RoboDK station: Tarea3Definitiva2_IsabellaCeballos.rdk

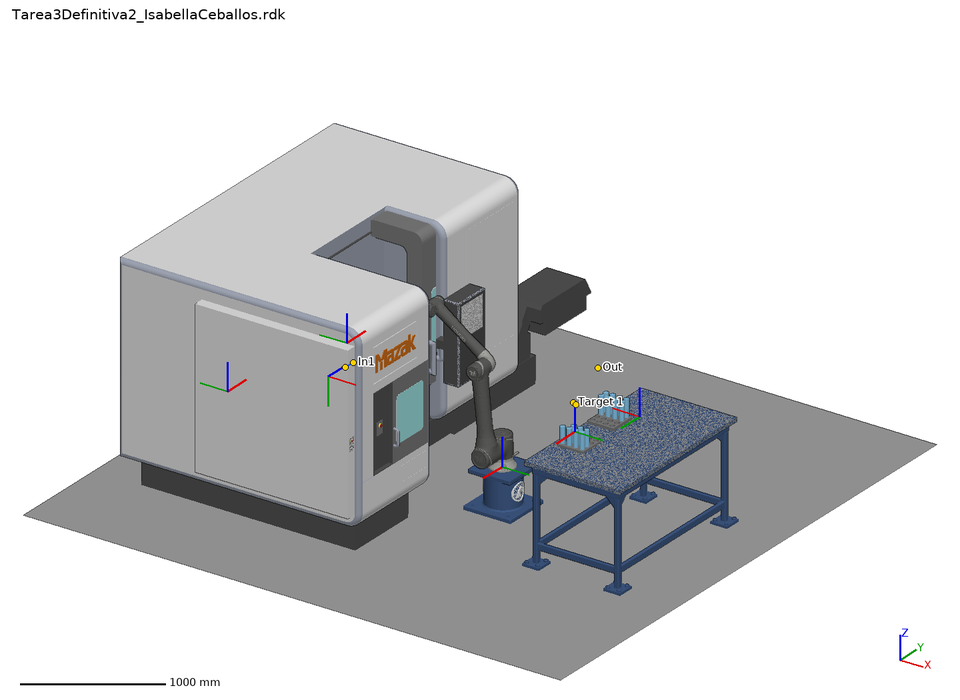
[picture v0: the station drawn from its stored meshes, robots at their saved joint values, targets as dots, program paths as lines]
Station Tarea3Definitiva2_IsabellaCeballos (saved by RoboDK 5.5.1). Poses are relative to the parent item; angles as X-Y-Z fixed-axis rotations.
Station parameters (name, value as stored): TAGS, ['Machine Tending', 'CNC']
  - frame Omron TM12X Base at (300, 0, 70) mm, rotated rx 0 ry 0 rz -90 deg
    - robot Omron TM12X: 6 axes, payload 12 kg, reach 1300 mm, repeatability 0.1 mm, weight 33.3 kg
        modified DH rows (alpha deg, a mm, theta deg, d mm): 0, 0, 0, 165.2; 90, 0, 90, 0; 0, 636.1, 0, 0; 0, 557.9, -90, 156.3; -90, 0, 0, 106; 90, 0, 180, 113.15
        joint limits [-360, -360, -163, -360, -360, -360] to [360, 360, 163, 360, 360, 360]; home [0, 0, 90, -90, 90, 0]; saved at [90.435, -6.151, -48.82, -37.474, -88.325, 69.903]
      - tool g1, TCP at (0, 0, 130) mm, size 134.4 x 157.6 x 75 mm
        - object Part 8 at (4.25, 9.04, 154.7) mm, rotated rx 177.54 ry -1.66 rz -69.47 deg, size 40 x 40 x 150 mm, geometry from Part.step
      - tool RobotiQ 2F-85 Gripper (Open), TCP at (0, 0, 130) mm, size 147.4 x 146.8 x 75 mm
    - object Pedestal H12in (Type 1) at (0, 10, -300) mm, size 400 x 400 x 304.8 mm, geometry from Pedestal-H12in-Type-1.sld
  - frame Mazak Lathe Base at (-1000, 0, 650) mm, rotated rx 0 ry 0 rz 90 deg
    - robot Mazak Lathe: 1 axes
        modified DH rows (alpha deg, a mm, theta deg, d mm): 0, 0, 0, 0 linear
        base shift (0, 0, 0) mm, rotated rx 0 ry 90 rz 0 deg
        joint limits [0] to [700]; home [0]; saved at [691]
    - frame Lathe at (-368.68, -104.77, -79.13) mm, rotated rx -90 ry 0 rz -90 deg
  - frame Input at (1010, -140, 590) mm, rotated rx 0 ry 0 rz -90 deg
    - object Part Matrix at (0, 0, 0) mm, size 220 x 220 x 25 mm, geometry from Part Matrix.step
    - target Target 1 (Cartesian target) at (-26.53, -36.52, 202.61) mm, rotated rx -177.37 ry 1.91 rz -69.45 deg; joints [247.43, -1, -72.52, -13.29, -90.61, 226.91] of Omron TM12X
    - object Part 6 at (137.5, 137.5, -20) mm, size 40 x 40 x 150 mm, geometry from Part.step
    - object Part 1 at (192.5, 192.5, -20) mm, size 40 x 40 x 150 mm, geometry from Part.step
    - object Part 5 at (137.5, 192.5, -20) mm, size 40 x 40 x 150 mm, geometry from Part.step
    - object Part 7 at (137.5, 82.5, -20) mm, size 40 x 40 x 150 mm, geometry from Part.step
    - object Part 4 at (192.5, 27.5, -20) mm, rotated rx 0 ry 0 rz -180 deg, size 40 x 40 x 150 mm, geometry from Part.step
    - object Part 3 at (192.5, 82.5, -20) mm, rotated rx 0 ry 0 rz -180 deg, size 40 x 40 x 150 mm, geometry from Part.step
    - object Part 2 at (192.5, 137.5, -20) mm, rotated rx 0 ry 0 rz -180 deg, size 40 x 40 x 150 mm, geometry from Part.step
    - target Home (Cartesian target) at (28, 28, 225) mm, rotated rx -177.37 ry 1.91 rz -69.45 deg; joints [245.421, -8.702, -61.622, -16.467, -90.498, 224.904] of Omron TM12X
    - target Out (Cartesian target) at (-404.5, -94.61, 298.15) mm, rotated rx 179.32 ry 1.81 rz -82.53 deg; joints [279.536, -58.254, 58.657, -88.574, -89.388, -87.935] of Omron TM12X
  - frame Output at (1250, 290, 600) mm, rotated rx 0 ry 0 rz -180 deg
    - object Part Matrix at (47.8, 28.1, 0) mm, size 220 x 220 x 25 mm, geometry from Part Matrix.step
    - object Part 16 at (75.39, 55.49, -8.13) mm, rotated rx 0 ry 0 rz 90 deg, size 40 x 40 x 150 mm, geometry from Part.step
    - object Part 15 at (132.39, 55.49, -8.13) mm, rotated rx 0 ry 0 rz 90 deg, size 40 x 40 x 150 mm, geometry from Part.step
    - object Part 14 at (189.39, 55.49, -8.13) mm, rotated rx 0 ry 0 rz 90 deg, size 40 x 40 x 150 mm, geometry from Part.step
    - object Part 13 at (246.39, 55.49, -8.13) mm, rotated rx 0 ry 0 rz 90 deg, size 40 x 40 x 150 mm, geometry from Part.step
    - object Part 12 at (75.39, 110.49, -8.13) mm, rotated rx 0 ry 0 rz 90 deg, size 40 x 40 x 150 mm, geometry from Part.step
    - object Part 11 at (132.39, 110.49, -8.13) mm, rotated rx 0 ry 0 rz 90 deg, size 40 x 40 x 150 mm, geometry from Part.step
    - object Part 10 at (189.39, 110.49, -8.13) mm, rotated rx 0 ry 0 rz 90 deg, size 40 x 40 x 150 mm, geometry from Part.step
    - object Part 9 at (246.39, 110.49, -8.13) mm, rotated rx 0 ry 0 rz 90 deg, size 40 x 40 x 150 mm, geometry from Part.step
  - frame World at (-2000, 0, 0) mm, rotated rx 0 ry 0 rz 90 deg
    - object Floor at (250, -1940, -230) mm, size 4500 x 4500 x 0 mm, geometry from Floor (2).sld
    - object Table 1400x800x800mm at (-340, -3360, 570) mm, size 1420 x 820 x 800 mm, geometry from Table-1400x800x800mm.sld
    - target OpenDoor (Cartesian target) at (700, -1000, 650) mm; joints [700] of Mazak Lathe
    - target CloseDoor (Cartesian target) at (0, -1000, 650) mm; joints [0] of Mazak Lathe
    - target In1 (Cartesian target) at (-137.95, -1150.25, 595.88) mm, rotated rx -86.34 ry 2.11 rz 94.34 deg; joints [77.244, -89.992, 25.646, 51.981, -342.661, 170.292] of Omron TM12X
    - target In2 (Cartesian target) at (-206.56, -1130.76, 584.67) mm, rotated rx -87.8 ry 7.87 rz 92.76 deg; joints [-84.147, 66.082, 6.025, 75.079, -175.968, 40.623] of Omron TM12X
  - program atach (1 instructions, listed below)
  - program detach (1 instructions, listed below)
  - program init (1 instructions, listed below)
  - program OpenDoor (2 instructions, listed below)
  - program CloseDoor (2 instructions, listed below)
  - program GoHome (3 instructions, listed below)
  - program Go_Out (3 instructions, listed below)
  - program Main_Program (496 instructions, listed below)
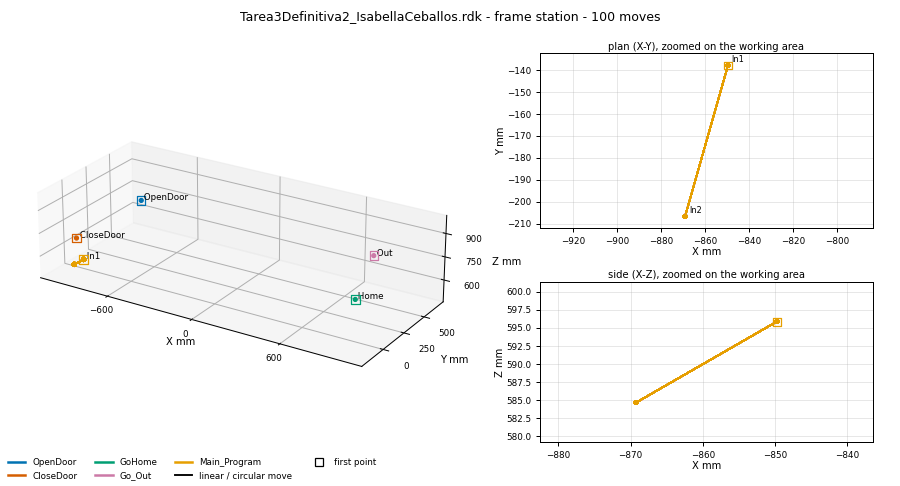
[picture p0: tool path of Tarea3Definitiva2_IsabellaCeballos.rdk in frame station, 100 of 276 moves have a stored position in this frame; points joined in program order, loops and branches not executed]

--- program atach (robot Omron TM12X) ---
  Adjuntar a g1

--- program detach (robot Omron TM12X) ---
  Separar de g1

--- program init (robot Omron TM12X) ---
  Reemplazar objetos

--- program OpenDoor (robot Mazak Lathe) ---
  Est. Ref.: World
  MoveJ (OpenDoor)

--- program CloseDoor (robot Mazak Lathe) ---
  Est. Ref.: World
  MoveJ (CloseDoor)

--- program GoHome (robot Omron TM12X) ---
  Est. Ref.: Input
  Est. herr: g1
  MoveJ (Home)

--- program Go_Out (robot Omron TM12X) ---
  Est. Ref.: Input
  Est. herr: g1
  MoveJ (Out)

--- program Main_Program (robot Omron TM12X) ---
  Est. Ref.: Input
  MoveJ (Auto Up_Pick 1) [its target is no longer in the station]
  MoveL (Auto Pick 1) [its target is no longer in the station]
  Llamar atach
  MoveL (Auto Up_Pick 1) [its target is no longer in the station]
  MoveL (Auto Transition 1) [its target is no longer in the station]
  MoveJ (Auto Transition 2) [its target is no longer in the station]
  Llamar OpenDoor
  Est. Ref.: World
  MoveJ (In1)
  MoveL (In2)
  Llamar detach
  MoveL (In1)
  Est. Ref.: Input
  MoveJ (Auto Transition 2) [its target is no longer in the station]
  Llamar CloseDoor
  Llamar OpenDoor
  Est. Ref.: World
  MoveJ (In1)
  MoveL (In2)
  Llamar atach
  MoveL (In1)
  Est. Ref.: Input
  MoveJ (Auto Transition 2) [its target is no longer in the station]
  Llamar CloseDoor
  MoveL (Auto Transition 1) [its target is no longer in the station]
  Llamar Go_Out
  MoveJ (Auto Drop_Up 1) [its target is no longer in the station]
  MoveL (Auto Drop 1) [its target is no longer in the station]
  Llamar detach
  MoveL (Auto Drop_Up 1) [its target is no longer in the station]
  Est. Ref.: Input
  MoveJ (Auto Up_Pick 2) [its target is no longer in the station]
  MoveL (Auto Pick 2) [its target is no longer in the station]
  Llamar atach
  MoveL (Auto Up_Pick 2) [its target is no longer in the station]
  MoveL (Auto Transition 1) [its target is no longer in the station]
  MoveJ (Auto Transition 2) [its target is no longer in the station]
  Llamar OpenDoor
  Est. Ref.: World
  MoveJ (In1)
  MoveL (In2)
  Llamar detach
  MoveL (In1)
  Est. Ref.: Input
  MoveJ (Auto Transition 2) [its target is no longer in the station]
  Llamar CloseDoor
  Llamar OpenDoor
  Est. Ref.: World
  MoveJ (In1)
  MoveL (In2)
  Llamar atach
  MoveL (In1)
  Est. Ref.: Input
  MoveJ (Auto Transition 2) [its target is no longer in the station]
  Llamar CloseDoor
  MoveL (Auto Transition 1) [its target is no longer in the station]
  Llamar Go_Out
  MoveJ (Auto Drop_Up 2) [its target is no longer in the station]
  MoveL (Auto Drop 2) [its target is no longer in the station]
  Llamar detach
  MoveL (Auto Drop_Up 2) [its target is no longer in the station]
  Est. Ref.: Input
  MoveJ (Auto Up_Pick 3) [its target is no longer in the station]
  MoveL (Auto Pick 3) [its target is no longer in the station]
  Llamar atach
  MoveL (Auto Up_Pick 3) [its target is no longer in the station]
  MoveL (Auto Transition 1) [its target is no longer in the station]
  MoveJ (Auto Transition 2) [its target is no longer in the station]
  Llamar OpenDoor
  Est. Ref.: World
  MoveJ (In1)
  MoveL (In2)
  Llamar detach
  MoveL (In1)
  Est. Ref.: Input
  MoveJ (Auto Transition 2) [its target is no longer in the station]
  Llamar CloseDoor
  Llamar OpenDoor
  Est. Ref.: World
  MoveJ (In1)
  MoveL (In2)
  Llamar atach
  MoveL (In1)
  Est. Ref.: Input
  MoveJ (Auto Transition 2) [its target is no longer in the station]
  Llamar CloseDoor
  MoveL (Auto Transition 1) [its target is no longer in the station]
  Llamar Go_Out
  MoveJ (Auto Drop_Up 3) [its target is no longer in the station]
  MoveL (Auto Drop 3) [its target is no longer in the station]
  Llamar detach
  MoveL (Auto Drop_Up 3) [its target is no longer in the station]
  Est. Ref.: Input
  MoveJ (Auto Up_Pick 4) [its target is no longer in the station]
  MoveL (Auto Pick 4) [its target is no longer in the station]
  Llamar atach
  MoveL (Auto Up_Pick 4) [its target is no longer in the station]
  MoveL (Auto Transition 1) [its target is no longer in the station]
  MoveJ (Auto Transition 2) [its target is no longer in the station]
  Llamar OpenDoor
  Est. Ref.: World
  MoveJ (In1)
  MoveL (In2)
  Llamar detach
  MoveL (In1)
  Est. Ref.: Input
  MoveJ (Auto Transition 2) [its target is no longer in the station]
  Llamar CloseDoor
  Llamar OpenDoor
  Est. Ref.: World
  MoveJ (In1)
  MoveL (In2)
  Llamar atach
  MoveL (In1)
  Est. Ref.: Input
  MoveJ (Auto Transition 2) [its target is no longer in the station]
  Llamar CloseDoor
  MoveL (Auto Transition 1) [its target is no longer in the station]
  Llamar Go_Out
  MoveJ (Auto Drop_Up 4) [its target is no longer in the station]
  MoveL (Auto Drop 4) [its target is no longer in the station]
  Llamar detach
  MoveL (Auto Drop_Up 4) [its target is no longer in the station]
  Est. Ref.: Input
  MoveJ (Auto Up_Pick 5) [its target is no longer in the station]
  MoveL (Auto Pick 5) [its target is no longer in the station]
  Llamar atach
  MoveL (Auto Up_Pick 5) [its target is no longer in the station]
  MoveL (Auto Transition 1) [its target is no longer in the station]
  MoveJ (Auto Transition 2) [its target is no longer in the station]
  Llamar OpenDoor
  Est. Ref.: World
  MoveJ (In1)
  MoveL (In2)
  Llamar detach
  MoveL (In1)
  Est. Ref.: Input
  MoveJ (Auto Transition 2) [its target is no longer in the station]
  Llamar CloseDoor
  Llamar OpenDoor
  Est. Ref.: World
  MoveJ (In1)
  MoveL (In2)
  Llamar atach
  MoveL (In1)
  Est. Ref.: Input
  MoveJ (Auto Transition 2) [its target is no longer in the station]
  Llamar CloseDoor
  MoveL (Auto Transition 1) [its target is no longer in the station]
  Llamar Go_Out
  MoveJ (Auto Drop_Up 5) [its target is no longer in the station]
  MoveL (Auto Drop 5) [its target is no longer in the station]
  Llamar detach
  MoveL (Auto Drop_Up 5) [its target is no longer in the station]
  Est. Ref.: Input
  MoveJ (Auto Up_Pick 6) [its target is no longer in the station]
  MoveL (Auto Pick 6) [its target is no longer in the station]
  Llamar atach
  MoveL (Auto Up_Pick 6) [its target is no longer in the station]
  MoveL (Auto Transition 1) [its target is no longer in the station]
  MoveJ (Auto Transition 2) [its target is no longer in the station]
  Llamar OpenDoor
  Est. Ref.: World
  MoveJ (In1)
  MoveL (In2)
  Llamar detach
  MoveL (In1)
  Est. Ref.: Input
  MoveJ (Auto Transition 2) [its target is no longer in the station]
  Llamar CloseDoor
  Llamar OpenDoor
  Est. Ref.: World
  MoveJ (In1)
  MoveL (In2)
  Llamar atach
  MoveL (In1)
  Est. Ref.: Input
  MoveJ (Auto Transition 2) [its target is no longer in the station]
  Llamar CloseDoor
  MoveL (Auto Transition 1) [its target is no longer in the station]
  Llamar Go_Out
  MoveJ (Auto Drop_Up 6) [its target is no longer in the station]
  MoveL (Auto Drop 6) [its target is no longer in the station]
  Llamar detach
  MoveL (Auto Drop_Up 6) [its target is no longer in the station]
  Est. Ref.: Input
  MoveJ (Auto Up_Pick 7) [its target is no longer in the station]
  MoveL (Auto Pick 7) [its target is no longer in the station]
  Llamar atach
  MoveL (Auto Up_Pick 7) [its target is no longer in the station]
  MoveL (Auto Transition 1) [its target is no longer in the station]
  MoveJ (Auto Transition 2) [its target is no longer in the station]
  Llamar OpenDoor
  Est. Ref.: World
  MoveJ (In1)
  MoveL (In2)
  Llamar detach
  MoveL (In1)
  Est. Ref.: Input
  MoveJ (Auto Transition 2) [its target is no longer in the station]
  Llamar CloseDoor
  Llamar OpenDoor
  Est. Ref.: World
  MoveJ (In1)
  MoveL (In2)
  Llamar atach
  MoveL (In1)
  Est. Ref.: Input
  MoveJ (Auto Transition 2) [its target is no longer in the station]
  Llamar CloseDoor
  MoveL (Auto Transition 1) [its target is no longer in the station]
  Llamar Go_Out
  MoveJ (Auto Drop_Up 7) [its target is no longer in the station]
  MoveL (Auto Drop 7) [its target is no longer in the station]
  Llamar detach
  MoveL (Auto Drop_Up 7) [its target is no longer in the station]
  Est. Ref.: Input
  MoveJ (Auto Up_Pick 8) [its target is no longer in the station]
  MoveL (Auto Pick 8) [its target is no longer in the station]
  Llamar atach
  MoveL (Auto Up_Pick 8) [its target is no longer in the station]
  MoveL (Auto Transition 1) [its target is no longer in the station]
  MoveJ (Auto Transition 2) [its target is no longer in the station]
  Llamar OpenDoor
  Est. Ref.: World
  MoveJ (In1)
  MoveL (In2)
  Llamar detach
  MoveL (In1)
  Est. Ref.: Input
  MoveJ (Auto Transition 2) [its target is no longer in the station]
  Llamar CloseDoor
  Llamar OpenDoor
  Est. Ref.: World
  MoveJ (In1)
  MoveL (In2)
  Llamar atach
  MoveL (In1)
  Est. Ref.: Input
  MoveJ (Auto Transition 2) [its target is no longer in the station]
  Llamar CloseDoor
  MoveL (Auto Transition 1) [its target is no longer in the station]
  Llamar Go_Out
  MoveJ (Auto Drop_Up 8) [its target is no longer in the station]
  MoveL (Auto Drop 8) [its target is no longer in the station]
  Llamar detach
  MoveL (Auto Drop_Up 8) [its target is no longer in the station]
  Est. Ref.: Input
  MoveJ (Auto Up_Pick 9) [its target is no longer in the station]
  MoveL (Auto Pick 9) [its target is no longer in the station]
  Llamar atach
  MoveL (Auto Up_Pick 9) [its target is no longer in the station]
  MoveL (Auto Transition 1) [its target is no longer in the station]
  MoveJ (Auto Transition 2) [its target is no longer in the station]
  Llamar OpenDoor
  Est. Ref.: World
  MoveJ (In1)
  MoveL (In2)
  Llamar detach
  MoveL (In1)
  Est. Ref.: Input
  MoveJ (Auto Transition 2) [its target is no longer in the station]
  Llamar CloseDoor
  Llamar OpenDoor
  Est. Ref.: World
  MoveJ (In1)
  MoveL (In2)
  Llamar atach
  MoveL (In1)
  Est. Ref.: Input
  MoveJ (Auto Transition 2) [its target is no longer in the station]
  Llamar CloseDoor
  MoveL (Auto Transition 1) [its target is no longer in the station]
  Llamar Go_Out
  MoveJ (Auto Drop_Up 9) [its target is no longer in the station]
  MoveL (Auto Drop 9) [its target is no longer in the station]
  Llamar detach
  MoveL (Auto Drop_Up 9) [its target is no longer in the station]
  Est. Ref.: Input
  MoveJ (Auto Up_Pick 10) [its target is no longer in the station]
  MoveL (Auto Pick 10) [its target is no longer in the station]
  Llamar atach
  MoveL (Auto Up_Pick 10) [its target is no longer in the station]
  MoveL (Auto Transition 1) [its target is no longer in the station]
  MoveJ (Auto Transition 2) [its target is no longer in the station]
  Llamar OpenDoor
  Est. Ref.: World
  MoveJ (In1)
  MoveL (In2)
  Llamar detach
  MoveL (In1)
  Est. Ref.: Input
  MoveJ (Auto Transition 2) [its target is no longer in the station]
  Llamar CloseDoor
  Llamar OpenDoor
  Est. Ref.: World
  MoveJ (In1)
  MoveL (In2)
  Llamar atach
  MoveL (In1)
  Est. Ref.: Input
  MoveJ (Auto Transition 2) [its target is no longer in the station]
  Llamar CloseDoor
  MoveL (Auto Transition 1) [its target is no longer in the station]
  Llamar Go_Out
  MoveJ (Auto Drop_Up 10) [its target is no longer in the station]
  MoveL (Auto Drop 10) [its target is no longer in the station]
  Llamar detach
  MoveL (Auto Drop_Up 10) [its target is no longer in the station]
  Est. Ref.: Input
  MoveJ (Auto Up_Pick 11) [its target is no longer in the station]
  MoveL (Auto Pick 11) [its target is no longer in the station]
  Llamar atach
  MoveL (Auto Up_Pick 11) [its target is no longer in the station]
  MoveL (Auto Transition 1) [its target is no longer in the station]
  MoveJ (Auto Transition 2) [its target is no longer in the station]
  Llamar OpenDoor
  Est. Ref.: World
  MoveJ (In1)
  MoveL (In2)
  Llamar detach
  MoveL (In1)
  Est. Ref.: Input
  MoveJ (Auto Transition 2) [its target is no longer in the station]
  Llamar CloseDoor
  Llamar OpenDoor
  Est. Ref.: World
  MoveJ (In1)
  MoveL (In2)
  Llamar atach
  MoveL (In1)
  Est. Ref.: Input
  MoveJ (Auto Transition 2) [its target is no longer in the station]
  Llamar CloseDoor
  MoveL (Auto Transition 1) [its target is no longer in the station]
  Llamar Go_Out
  MoveJ (Auto Drop_Up 11) [its target is no longer in the station]
  MoveL (Auto Drop 11) [its target is no longer in the station]
  Llamar detach
  MoveL (Auto Drop_Up 11) [its target is no longer in the station]
  Est. Ref.: Input
  MoveJ (Auto Up_Pick 12) [its target is no longer in the station]
  MoveL (Auto Pick 12) [its target is no longer in the station]
  Llamar atach
  MoveL (Auto Up_Pick 12) [its target is no longer in the station]
  MoveL (Auto Transition 1) [its target is no longer in the station]
  MoveJ (Auto Transition 2) [its target is no longer in the station]
  Llamar OpenDoor
  Est. Ref.: World
  MoveJ (In1)
  MoveL (In2)
  Llamar detach
  MoveL (In1)
  Est. Ref.: Input
  MoveJ (Auto Transition 2) [its target is no longer in the station]
  Llamar CloseDoor
  Llamar OpenDoor
  Est. Ref.: World
  MoveJ (In1)
  MoveL (In2)
  Llamar atach
  MoveL (In1)
  Est. Ref.: Input
  MoveJ (Auto Transition 2) [its target is no longer in the station]
  Llamar CloseDoor
  MoveL (Auto Transition 1) [its target is no longer in the station]
  Llamar Go_Out
  MoveJ (Auto Drop_Up 12) [its target is no longer in the station]
  MoveL (Auto Drop 12) [its target is no longer in the station]
  Llamar detach
  MoveL (Auto Drop_Up 12) [its target is no longer in the station]
  Est. Ref.: Input
  MoveJ (Auto Up_Pick 13) [its target is no longer in the station]
  MoveL (Auto Pick 13) [its target is no longer in the station]
  Llamar atach
  MoveL (Auto Up_Pick 13) [its target is no longer in the station]
  MoveL (Auto Transition 1) [its target is no longer in the station]
  MoveJ (Auto Transition 2) [its target is no longer in the station]
  Llamar OpenDoor
  Est. Ref.: World
  MoveJ (In1)
  MoveL (In2)
  Llamar detach
  MoveL (In1)
  Est. Ref.: Input
  MoveJ (Auto Transition 2) [its target is no longer in the station]
  Llamar CloseDoor
  Llamar OpenDoor
  Est. Ref.: World
  MoveJ (In1)
  MoveL (In2)
  Llamar atach
  MoveL (In1)
  Est. Ref.: Input
  MoveJ (Auto Transition 2) [its target is no longer in the station]
  Llamar CloseDoor
  MoveL (Auto Transition 1) [its target is no longer in the station]
  Llamar Go_Out
  MoveJ (Auto Drop_Up 13) [its target is no longer in the station]
  MoveL (Auto Drop 13) [its target is no longer in the station]
  Llamar detach
  MoveL (Auto Drop_Up 13) [its target is no longer in the station]
  Est. Ref.: Input
  MoveJ (Auto Up_Pick 14) [its target is no longer in the station]
  MoveL (Auto Pick 14) [its target is no longer in the station]
  Llamar atach
  MoveL (Auto Up_Pick 14) [its target is no longer in the station]
  MoveL (Auto Transition 1) [its target is no longer in the station]
  MoveJ (Auto Transition 2) [its target is no longer in the station]
  Llamar OpenDoor
  Est. Ref.: World
  MoveJ (In1)
  MoveL (In2)
  Llamar detach
  MoveL (In1)
  Est. Ref.: Input
  MoveJ (Auto Transition 2) [its target is no longer in the station]
  Llamar CloseDoor
  Llamar OpenDoor
  Est. Ref.: World
  MoveJ (In1)
  MoveL (In2)
  Llamar atach
  MoveL (In1)
  Est. Ref.: Input
  MoveJ (Auto Transition 2) [its target is no longer in the station]
  Llamar CloseDoor
  MoveL (Auto Transition 1) [its target is no longer in the station]
  Llamar Go_Out
  MoveJ (Auto Drop_Up 14) [its target is no longer in the station]
  MoveL (Auto Drop 14) [its target is no longer in the station]
  Llamar detach
  MoveL (Auto Drop_Up 14) [its target is no longer in the station]
  Est. Ref.: Input
  MoveJ (Auto Up_Pick 15) [its target is no longer in the station]
  MoveL (Auto Pick 15) [its target is no longer in the station]
  Llamar atach
  MoveL (Auto Up_Pick 15) [its target is no longer in the station]
  MoveL (Auto Transition 1) [its target is no longer in the station]
  MoveJ (Auto Transition 2) [its target is no longer in the station]
  Llamar OpenDoor
  Est. Ref.: World
  MoveJ (In1)
  MoveL (In2)
  Llamar detach
  MoveL (In1)
  Est. Ref.: Input
  MoveJ (Auto Transition 2) [its target is no longer in the station]
  Llamar CloseDoor
  Llamar OpenDoor
  Est. Ref.: World
  MoveJ (In1)
  MoveL (In2)
  Llamar atach
  MoveL (In1)
  Est. Ref.: Input
  MoveJ (Auto Transition 2) [its target is no longer in the station]
  Llamar CloseDoor
  MoveL (Auto Transition 1) [its target is no longer in the station]
  Llamar Go_Out
  MoveJ (Auto Drop_Up 15) [its target is no longer in the station]
  MoveL (Auto Drop 15) [its target is no longer in the station]
  Llamar detach
  MoveL (Auto Drop_Up 15) [its target is no longer in the station]
  Est. Ref.: Input
  MoveJ (Auto Up_Pick 16) [its target is no longer in the station]
  MoveL (Auto Pick 16) [its target is no longer in the station]
  Llamar atach
  MoveL (Auto Up_Pick 16) [its target is no longer in the station]
  MoveL (Auto Transition 1) [its target is no longer in the station]
  MoveJ (Auto Transition 2) [its target is no longer in the station]
  Llamar OpenDoor
  Est. Ref.: World
  MoveJ (In1)
  MoveL (In2)
  Llamar detach
  MoveL (In1)
  Est. Ref.: Input
  MoveJ (Auto Transition 2) [its target is no longer in the station]
  Llamar CloseDoor
  Llamar OpenDoor
  Est. Ref.: World
  MoveJ (In1)
  MoveL (In2)
  Llamar atach
  MoveL (In1)
  Est. Ref.: Input
  MoveJ (Auto Transition 2) [its target is no longer in the station]
  Llamar CloseDoor
  MoveL (Auto Transition 1) [its target is no longer in the station]
  Llamar Go_Out
  MoveJ (Auto Drop_Up 16) [its target is no longer in the station]
  MoveL (Auto Drop 16) [its target is no longer in the station]
  Llamar detach
  MoveL (Auto Drop_Up 16) [its target is no longer in the station]
